{attribute 'GeneratedUsingTerminal: EP6002-0002-0016'}
{attribute addProperty BoxType "EP6002-0002-0016"}
{attribute addProperty Id "CtrlAT %Q*WORD2Data_OutAT %Q*ARRAY[0..21] OF USINT22"}
{attribute addProperty CRC "1305863315"}
{attribute addProperty Size "24"}
TYPE COM_Outputs_Channel_B336F4EE :
STRUCT
	{attribute addProperty Name "Ctrl"}
	Ctrl AT %Q* : WORD;
	{attribute addProperty Name "Data_Out"}
	Data_Out AT %Q* : ARRAY[0..21] OF USINT;
END_STRUCT
END_TYPE

(* stored: Version 1.2.0.0, ProductVersion 3.1.4024.9
   DUT COM_Outputs_Channel_B336F4EE: Id {c1282641-05e4-4c28-b67a-80d2dcc5821a} *)
